(* LS Electric XG5000 project: XMC_AC_Drive_Ctrl_FB *)
(* PLC LSPLC *)
(* module base 0 slot 0: Input/Output Module:XMC-DN24 (DC 24V Input 8Points/TR output 16Points) *)
(* module base 0 slot 1: Internal Analog Input/Output:XMF-AH04E (A/D voltage/current 2 channels, D/A voltage 2 channels) *)
(* task Periodic Task: Kind=2 *)
(* task Initialization Task: Kind=1 *)
(* task NC Program: Kind=6 *)

FUNCTION_BLOCK XMC_AC_Drive_Ctrl_FB
(* This funciton block is used to provide ease of use for controlling EtherCAT AC drives with the XMC *)
VAR_IN_OUT
    Axis : UINT; (* Axis number of the AC drive. *)
END_VAR
VAR_INPUT
    Enable_Drive : BOOL; (* 0: Disable the drive;  1: Enable drive for operation / Motion will resume when drive is re-enabled. *)
    Quick_Stop : BOOL; (* 0: Motion not stopped;  1: Quick Stop the drive. / Motion will continue when reset back to 0. *)
    Change_Velocity : BOOL; (* Will change AC drive velocity on rising edge. *)
    Target_Velocity : INT; (* Target velocity of the AC drive in RPM. *)
    Reset_Fault : BOOL; (* Used to reset a fault *)
END_VAR
VAR_OUTPUT
    Drive_Enabled : BOOL; (* Status that the drive is Enabled *)
    Current_Velocity : INT; (* Current speed of the AC drive in RPM *)
    Drive_Faulted : BOOL; (* Status that the Drive is faulted *)
END_VAR
VAR CONSTANT
    Fault_Reaction_Active : USINT := 70; (* State status of Fault reaction active. *)
    Fault_State : USINT := 60; (* State status of Drive fault *)
    Not_Ready_To_Switch_On : USINT := 0; (* State status for Not Ready to switch on *)
    Operation_Enabled : USINT := 40; (* State status of Operation enabled *)
    Quick_Stop_Active : USINT := 50; (* State status of Quick stop active *)
    Ready_To_Switch_On : USINT := 20; (* State status of Ready to Switch On *)
    Switched_On : USINT := 30; (* State status of Switched on *)
    Switch_On_Disabled : USINT := 10; (* State status of Switch on disabled *)
END_VAR
VAR
    Previous_Change_Velocity : BOOL; (* history storage for change in velocity command *)
    Read_Status1 : LS_INVERTERSTATUS1; (* local function block for reading AC drive status *)
    Read_Status2 : LS_INVERTERSTATUS2; (* local funciton block for reading AC drive status *)
    Read_Velocity : LS_INVERTERREADVEL; (* local funciton block for reading drive velocity *)
    State : USINT := 0; (* State variable for controlling the AC drive *)
    Write_Control_Word : LS_INVERTERCONTROL; (* local function block for writing control word to the AC drive *)
    Write_Velocity : LS_INVERTERWRITEVEL; (* local function block for writing drive velocity *)
END_VAR
(* 
AutomationDirect.com has provided this code for convenience. This sample code is provided "as-is" with no expressed or implied warranty. 
 If the end user includes any of the sample code (in whole or part), it is the user's responsibility to completely modify, integrate, and test any code to ensure it meets all system and 
 safety requirements for the intended application or system.
 *)
 
 //If AC drive is faulted then move state machine to faulted state
 IF (Drive_Faulted) THEN
 	State := Fault_State;
 END_IF;	
 
 //Change previous velocity storage state if command to change velocity is set to FALSE
 IF (Change_Velocity = FALSE) THEN
 	Previous_Change_Velocity := FALSE;
 	Write_Velocity.Execute := FALSE;
 END_IF;

//State Machine for AC Drive control
CASE State OF
	
	//Drive starts in Not ready to switch on.  Wait for Drive to be in Switch On Disabled.
	0:
		IF (Enable_Drive = TRUE) THEN   //(Read_Status1.SwOnDisable) THEN
			State := Switch_On_Disabled;
		END_IF;
		
	//Switch On Disabled state	
	10: 	
		IF (Enable_Drive = TRUE) AND (Quick_Stop = FALSE) THEN
			Write_Control_Word.SwitchOn := FALSE;
			Write_Control_Word.VoltageEn := TRUE;
			Write_Control_Word.QuickStop := TRUE;
			Write_Control_Word.EnableOP := FALSE;
			
			Write_Control_Word.Execute :=  TRUE;
			
			//Move state machine to Ready To Switch On state
			IF (Read_Status1.RdySwitchOn) AND (Write_Control_Word.Done) THEN
				Write_Control_Word.Execute := FALSE;
				State :=  Ready_To_Switch_On;
			END_IF;
					
		ELSIF (Enable_Drive = FALSE) THEN		
			Write_Control_Word.SwitchOn := FALSE;
			Write_Control_Word.VoltageEn := FALSE;
			Write_Control_Word.QuickStop := FALSE;
			Write_Control_Word.EnableOP := FALSE;
			Write_Control_Word.Execute :=  FALSE;
		END_IF;	
		
	//Ready to Switch On State	
	20:
		IF (Enable_Drive = TRUE) THEN
			Write_Control_Word.SwitchOn := TRUE;
			Write_Control_Word.VoltageEn := TRUE;
			Write_Control_Word.QuickStop := TRUE;
			Write_Control_Word.EnableOP := FALSE;
			
			Write_Control_Word.Execute :=  TRUE;
			
			//Move state machine to Ready To Switch On state
			IF (Read_Status1.SwitchedOn) AND (Write_Control_Word.Done) THEN
				Write_Control_Word.Execute := FALSE;
				State :=  Switched_On;
			END_IF;
		
		
		ELSIF (Enable_Drive = FALSE) THEN
			Write_Control_Word.SwitchOn := FALSE;
			Write_Control_Word.VoltageEn := FALSE;
			Write_Control_Word.QuickStop := FALSE;
			Write_Control_Word.EnableOP := FALSE;
			
			Write_Control_Word.Execute :=  TRUE;
			
			//Move state machine to Quick Stop Active state
			IF (Read_Status1.SwOnDisable = FALSE) AND (Write_Control_Word.Done) THEN
				Write_Control_Word.Execute := FALSE;
				State :=  Switch_On_Disabled;
			END_IF;	
			
		END_IF;		
		
		
	//Switched On State	
	30:	
		IF (Enable_Drive = TRUE) THEN
			Write_Control_Word.SwitchOn := TRUE;
			Write_Control_Word.VoltageEn := TRUE;
			Write_Control_Word.QuickStop := TRUE;
			Write_Control_Word.EnableOP := TRUE;
			
			Write_Control_Word.Execute :=  TRUE;
			
			//Move state machine to Ready To Switch On state
			IF (Read_Status1.OpEn) AND (Write_Control_Word.Done) THEN
				Write_Control_Word.Execute := FALSE;
				State :=  Operation_Enabled;
			END_IF;
		
		ELSIF (Enable_Drive = FALSE) THEN
			Write_Control_Word.SwitchOn := FALSE;
			Write_Control_Word.VoltageEn := FALSE;
			Write_Control_Word.QuickStop := FALSE;
			Write_Control_Word.EnableOP := FALSE;
			
			Write_Control_Word.Execute :=  TRUE;
			
			//Move state machine to Quick Stop Active state
			IF (Read_Status1.SwOnDisable = FALSE) AND (Write_Control_Word.Done) THEN
				Write_Control_Word.Execute := FALSE;
				State :=  Switch_On_Disabled;
			END_IF;	
			
		END_IF;			
		
	//Operation Enabled state	
	40:		
		//disable the drive
		IF (Enable_Drive =  FALSE) THEN
			Write_Control_Word.SwitchOn := FALSE;
			Write_Control_Word.VoltageEn := FALSE;
			Write_Control_Word.QuickStop := FALSE;
			Write_Control_Word.EnableOP := FALSE;
			
			Write_Control_Word.Execute :=  TRUE;
			
			//Move state machine to Quick Stop Active state
			IF (Read_Status1.SwOnDisable = FALSE) AND (Write_Control_Word.Done) THEN
				Write_Control_Word.Execute := FALSE;
				State :=  Switch_On_Disabled;
			END_IF;
				
		//stop motion
		ELSIF (Quick_Stop =  TRUE) THEN
			Write_Control_Word.SwitchOn := TRUE;
			Write_Control_Word.VoltageEn := TRUE;
			Write_Control_Word.QuickStop := FALSE;
			Write_Control_Word.EnableOP := TRUE;
			
			Write_Control_Word.Execute :=  TRUE;
			
			//Move state machine to Quick Stop Active state
			IF (Read_Status2.QuickStop) AND (Write_Control_Word.Done) THEN
				Write_Control_Word.Execute := FALSE;
				State :=  Quick_Stop_Active;
			END_IF;
			
		//Change drive velocity	
		ELSIF (Change_Velocity = TRUE) AND (Previous_Change_Velocity = FALSE) THEN
			Write_Velocity.Execute := TRUE;	
			
			IF (Write_Velocity.Done) THEN
				Write_Velocity.Execute := FALSE;
				Previous_Change_Velocity := TRUE;
			END_IF;	

	
		END_IF; //end main if statement of Operation enable state
	
	//Quick Stop Active state
	50:
		//disable the drive
		IF (Quick_Stop =  FALSE) THEN
			Write_Control_Word.SwitchOn := FALSE;
			Write_Control_Word.VoltageEn := FALSE;
			Write_Control_Word.QuickStop := FALSE;
			Write_Control_Word.EnableOP := FALSE;
			
			Write_Control_Word.Execute :=  TRUE;
			
			//Move state machine to Quick Stop Active state
			IF (Read_Status1.SwOnDisable = TRUE) AND (Write_Control_Word.Done) THEN
				Write_Control_Word.Execute := FALSE;
				State :=  Switch_On_Disabled;
			END_IF;
		END_IF; //end main if in Quick stop active		
	
	//Fault state
	60:
		IF (Reset_Fault) THEN
			Write_Control_Word.SwitchOn := FALSE;
			Write_Control_Word.VoltageEn := FALSE;
			Write_Control_Word.QuickStop := FALSE;
			Write_Control_Word.EnableOP := FALSE;
			Write_Control_Word.FaultReset := TRUE;
			
			Write_Control_Word.Execute :=  TRUE;
			
			//Move state machine to Quick Stop Active state
			IF (Read_Status2.Fault = FALSE) AND (Write_Control_Word.Done) THEN
				Write_Control_Word.Execute := FALSE;
				Write_Control_Word.FaultReset := FALSE;
				State :=  Switch_On_Disabled;
			END_IF;
		END_IF;	
	
END_CASE; // end state machine



//local AC drive function block calls
Write_Control_Word(Execute:=Write_Control_Word.Execute, Axis:=Axis, SwitchOn:=Write_Control_Word.SwitchOn, VoltageEn:=Write_Control_Word.VoltageEn, QuickStop:=Write_Control_Word.QuickStop, EnableOP:=Write_Control_Word.EnableOP, EnableRamp:=Write_Control_Word.EnableRamp, UnlockRamp:=Write_Control_Word.UnlockRamp, ReferenceRamp:=Write_Control_Word.ReferenceRamp, FaultReset:=Write_Control_Word.FaultReset, Halt:=Write_Control_Word.Halt);
Write_Velocity(Execute:=Write_Velocity.Execute, Axis:=Axis, TargetVel:=Target_Velocity);

Read_Status1(Enable:=Enable_Drive, Axis:=Axis, OpEn=>Drive_Enabled);
Read_Status2(Enable:=Enable_Drive, Axis:=Axis, Fault=>Drive_Faulted);
Read_Velocity(Enable:=TRUE, Axis:=Axis,  ActualVel=>Current_Velocity);
END_FUNCTION_BLOCK

PROGRAM NewProgram (* task: Scan Program *)
VAR
    AC_Drive_INST : XMC_AC_Drive_Ctrl_FB; (* function block to control an AC drive over EtherCAT *)
    Axis1 : UINT; (* Axis variable for Axis 1 *)
    Change_Velocity : BOOL; (* Command to change AC drive velocity *)
    Connect_Busy : BOOL; (* busy status for LS_Conncet *)
    Connect_Error : BOOL; (* error status for LS_Connect *)
    Connect_ErrorID : WORD; (* error identification for LS_Connect *)
    Current_Velocity : INT; (* current Velocity of the AC drive *)
    Disconnect_Busy : BOOL; (* busy status for LS_Disconnect *)
    Disconnect_Error : BOOL; (* Error status for LS_Disconnect *)
    Disconnect_ErrorID : WORD; (* error identification for LS_DIsconnect *)
    Drive_Enabled : BOOL; (* Status that AC drive is enabled *)
    Drive_Faulted : BOOL; (* status that the AC drive is faulted *)
    ECAT_Connect : LS_CONNECT; (* function block to connect EtherCAT network *)
    ECAT_Disconnect : LS_DISCONNECT; (* function block to disconnect the EtherCAT network *)
    Enable_Drive : BOOL; (* enable the AC Drive *)
    Execute_Connect : BOOL; (* Execute the connection of EtherCAT network *)
    Execute_Disconnect : BOOL; (* execute LS_Disconnect *)
    Quick_Stop : BOOL; (* stop AC drive motion. Motion will resume when set to '0'. *)
    Reset_Fault : BOOL; (* Command to reset an AC drive fault *)
    Target_Velocity : INT; (* Velocity in RPM to set to AC drive *)
END_VAR

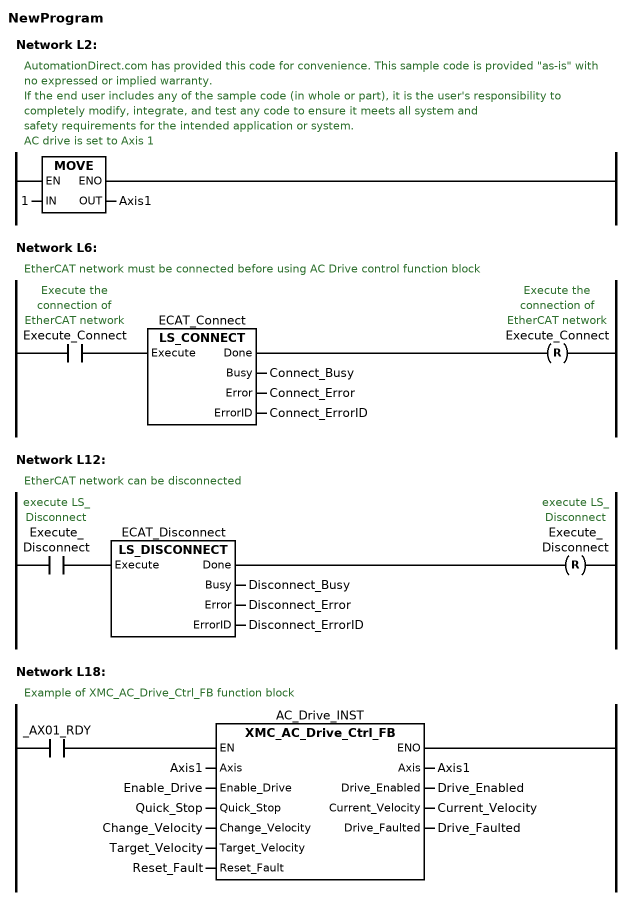
(* AutomationDirect.com has provided this code for convenience. This sample code is provided "as-is" with no expressed or implied warranty. / If the end user includes any of the sample code (in whole or part), it is the user's responsibility to completely modify, integrate, and test any code to ensure it meets all system and / safety requirements for the intended application or system. *)
(* AC drive is set to Axis 1 *)
(* Rung L2 *)
Axis1 := 1;
(* EtherCAT network must be connected before using AC Drive control function block *)
(* Rung L6 *)
ECAT_Connect(Execute := Execute_Connect, Busy => Connect_Busy, Error => Connect_Error, ErrorID => Connect_ErrorID);
IF ECAT_Connect.Done THEN Execute_Connect := FALSE; END_IF;
(* EtherCAT network can be disconnected *)
(* Rung L12 *)
ECAT_Disconnect(Execute := Execute_Disconnect, Busy => Disconnect_Busy, Error => Disconnect_Error, ErrorID => Disconnect_ErrorID);
IF ECAT_Disconnect.Done THEN Execute_Disconnect := FALSE; END_IF;
(* Example of XMC_AC_Drive_Ctrl_FB function block *)
(* Rung L18 *)
IF _AX01_RDY THEN
    AC_Drive_INST(Axis := Axis1, Enable_Drive := Enable_Drive, Quick_Stop := Quick_Stop, Change_Velocity := Change_Velocity, Target_Velocity := Target_Velocity, Reset_Fault := Reset_Fault, Axis => Axis1, Drive_Enabled => Drive_Enabled, Current_Velocity => Current_Velocity, Drive_Faulted => Drive_Faulted);
END_IF;
END_PROGRAM